Staubli VAL3: onF3Event.pgx

program onF3Event(bool x_bSave)
  local string l_sMessage
  local bool l_bYes
  local string l_sButton[2]
begin
  // look if the bButton is enable
  if bButton[2]
    //
    if !cycleStatus:bCycle and nIndexTool==0
      call language:message(l_sMessage,125)
      // get the yes_no button
      call language:getYesNo(l_sButton)
      // ask the question
      call use:yes_no(l_sMessage,l_sButton,l_bYes)
      if l_bYes
        call tcp:here()
        call language:message(l_sMessage,121)
        popUpMsg(l_sMessage)
        logMsg("[KERNEL] INTERFACE:Take the reference point")
        x_bSave=true
      endIf
    endIf
  endIf
end
